% RSLogix 500 project P7_SENSOR_CALIBRATOR.RSS, saved by version 8.30.00.16 %
PROJECT "UNTITLED"    % processor: Bul.1763 MicroLogix 1100 Series B %

PROGRAM FILES
  LAD 2   7 rungs

DATA FILES
  O0 OUTPUT  4 elements
  I1 INPUT  6 elements
  S2 STATUS  66 elements
  B3 BINARY  3 elements
  T4 TIMER  5 elements
  C5 COUNTER  1 elements
  R6 CONTROL  1 elements
  N7 INTEGER  6 elements
  F8 FLOAT  1 elements

LADDER 2
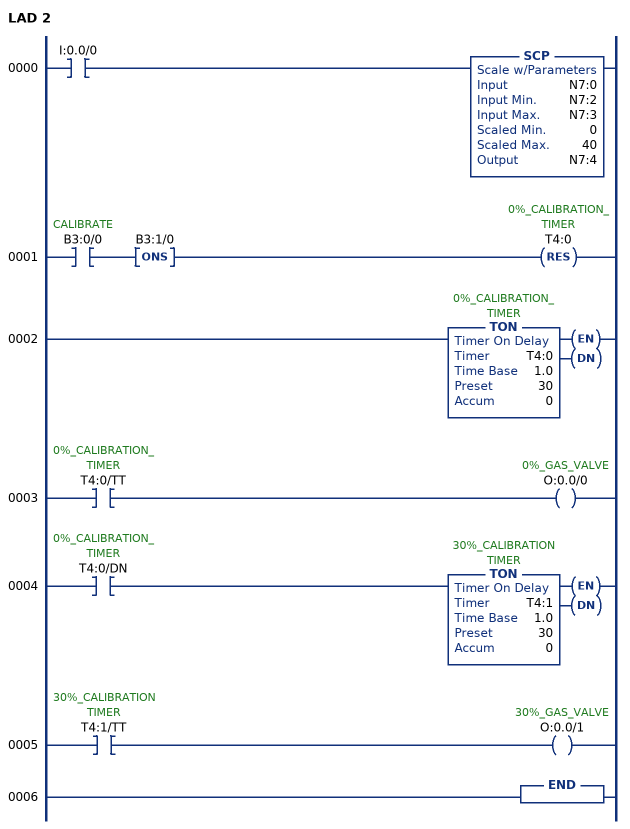
% Rung: 0 %
SOR XIC I:0.0/0 SCP N7:0 N7:2 N7:3 0 40 N7:4 EOR
%   N7:0  "O2_SENSOR_INP" %
%   N7:2  "O2_INPUT_MIN" %
%   N7:3  "O2_INPUT_MAX" %
% Rung: 1 %
SOR XIC B3:0/0 ONS B3:1/0 RES T4:0 EOR
%   B3:0/0  "CALIBRATE" %
%   T4:0  "0%_CALIBRATION_TIMER" %
% Rung: 2 %
SOR TON T4:0 1.0 30 0 EOR
%   T4:0  "0%_CALIBRATION_TIMER" %
% Rung: 3 %
SOR XIC T4:0/TT OTE O:0.0/0 EOR
%   T4:0  "0%_CALIBRATION_TIMER" %
%   O:0.0/0  "0%_GAS_VALVE" %
% Rung: 4 %
SOR XIC T4:0/DN TON T4:1 1.0 30 0 EOR
%   T4:0  "0%_CALIBRATION_TIMER" %
%   T4:1  "30%_CALIBRATION TIMER" %
% Rung: 5 %
SOR XIC T4:1/TT OTE O:0.0/1 EOR
%   T4:1  "30%_CALIBRATION TIMER" %
%   O:0.0/1  "30%_GAS_VALVE" %
% Rung: 6 %
SOR END EOR

OTHER DOCUMENTED ADDRESSES
  B3:1  "ONS"
  N7:1  "MEASURED_O2_CONCENTR ATION"

DATA TABLE (non-zero values as saved)
DATA T4
% .PRE .ACC %
% T4:0 % 30 0
% T4:1 % 30 0
DATA N7
% N7:0 % 0 0 0 16383 0 0
